FUNCTION_BLOCK REJECTION_COND (* Composite Function Block Type *)
  (* Standard: 61499-2 *)
  (* Version 0.2, 2003-12-05, JHC, Rockwell Automation, Renamed from NEWCOMPFB. *)
  (* Version 0.1, 2002-01-08, JHC, Rockwell Automation, Added DLY FB as example. *)
  (* Version 0.0, 2000-05-27, JHC, Rockwell Automation *)
  (* Compiler header: package fb.rt.student; *)
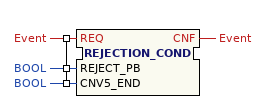
  EVENT_INPUT
    REQ WITH REJECT_PB, CNV5_END; (* Normal Execution Request *)
  END_EVENT
  EVENT_OUTPUT
    CNF; (* Execution Confirmation *)
  END_EVENT
  VAR_INPUT
    REJECT_PB : BOOL;
    CNV5_END : BOOL;
  END_VAR
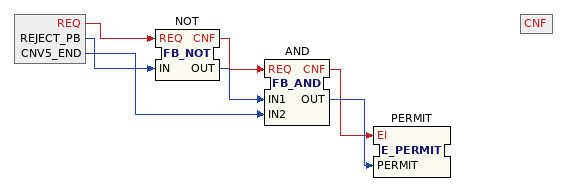
  FBS
    NOT : FB_NOT;
    AND : FB_AND;
    PERMIT : E_PERMIT;
  END_FBS
  EVENT_CONNECTIONS
    REQ TO NOT.REQ;
    NOT.CNF TO AND.REQ;
    AND.CNF TO PERMIT.EI;
  END_CONNECTIONS
  DATA_CONNECTIONS
    REJECT_PB TO NOT.IN;
    NOT.OUT TO AND.IN1;
    CNV5_END TO AND.IN2;
    AND.OUT TO PERMIT.PERMIT;
  END_CONNECTIONS
END_FUNCTION_BLOCK
